// TIA Portal V18 program export: 1 tag tables, 3 data types, 7 data blocks, 7 code blocks (in call order from the OBs), 0 instance data blocks

VAR_GLOBAL   // PLC tag table "DefaultTagTable"
   convRight AT %I0.0 : Bool;
   convLeft AT %I0.1 : Bool;
   manualMode AT %Q0.2 : Bool;
   automaticMode AT %Q0.3 : Bool;
END_VAR

TYPE "typeConvCmd"
TITLE = Conveyor command
VERSION : 0.1
//input Signals to Conv
   STRUCT
      enable : Bool;
      inputLigBeam : Bool;   // light beam on input of conveyor
      editLigBeam : Bool;   // light beam on edit station of brownie
      outputLigBeam : Bool;   // light beam on output of conveyor
      startConv : Bool;   // manual start of conveyor
      reset : Bool;   // reset of conveyor belt
      workStationDone : Bool;   // working station has done process
   END_STRUCT;

END_TYPE

TYPE "typeConvSig"
TITLE = Conveyor command / status signals
VERSION : 0.1
   STRUCT
      convIn : "typeConvCmd";
      convOut : "typeConvStat";
   END_STRUCT;

END_TYPE

TYPE "typeConvStat"
TITLE = conveyor status
VERSION : 0.1
//output signal of conveyors
   STRUCT
      valid : Bool;   // as output
      isRunning : Bool;   // conveyor is running
   END_STRUCT;

END_TYPE

DATA_BLOCK "InstConveyor"
{ S7_Optimized_Access := 'TRUE' }
VERSION : 0.1
NON_RETAIN
"Conveyor"

BEGIN

END_DATA_BLOCK

DATA_BLOCK "InstRoboter"
{ S7_Optimized_Access := 'TRUE' }
VERSION : 0.1
NON_RETAIN
"Robot"

BEGIN

END_DATA_BLOCK

DATA_BLOCK "InstSequencer"
{ S7_Optimized_Access := 'TRUE' }
VERSION : 0.1
NON_RETAIN
"Sequencer"

BEGIN
   BasicPosition.T_MAX := T#0MS;
   BasicPosition.T_WARN := T#0MS;
   StartConveyor.T_MAX := T#420MS;
   StartConveyor.T_WARN := T#385MS;
   MovePart.T_MAX := T#6S_408MS;
   MovePart.T_WARN := T#5S_874MS;
   GoToStation.T_MAX := T#3S_936MS;
   GoToStation.T_WARN := T#3S_608MS;
   Fill.T_MAX := T#3S_606MS;
   Fill.T_WARN := T#3S_305MS;
   GoToMagazine.T_MAX := T#3S_966MS;
   GoToMagazine.T_WARN := T#3S_635MS;
   RemovePart.T_MAX := T#4S_56MS;
   RemovePart.T_WARN := T#3S_718MS;
   ResetPositions.T_MAX := T#0MS;
   ResetPositions.T_WARN := T#0MS;
   ResetConveyor.T_MAX := T#0MS;
   ResetConveyor.T_WARN := T#0MS;

END_DATA_BLOCK

DATA_BLOCK "InstSimulation"
{ S7_Optimized_Access := 'TRUE' }
VERSION : 0.1
NON_RETAIN
"Simulation"

BEGIN

END_DATA_BLOCK

DATA_BLOCK "SeqData"
{ S7_Optimized_Access := 'TRUE' }
VERSION : 0.1
NON_RETAIN
   VAR 
      startButton : Bool;   // Start sequence
      ackSeq : Bool;   // Acknowledge sequence errors
      switchOffSeq : Bool;   // Stop sequence
      initSeq : Bool;   // Initialise sequence
      simulateError : Bool;   // Engine has fault (simulated)
      resetCrit : Bool;   // Reset sequence errors
      seqNumber : Int;   // Active sequence number
      error : Bool;   // Sequence has an error
      automaticMode : Bool;   // Sequence mode: automatic
      manualMode : Bool;   // Sequence mode: manual
      lightBeam1 : Bool;
      lightBeam2 : Bool;
      lightBeam3 : Bool;
      partInPos1 : Bool;   // Status part is in position 1
      partInPos2 : Bool;   // Status part is in position 2
      partInPos3 : Bool;   // Status part is in position 3
      robotFill : Bool;   // Command for robot to fill part
      robotGoToStation : Bool;   // Command for robot to go to station
      robotGoToMagazine : Bool;   // Command for robot to go to magazine
      robotOnStation : Bool;   // Status robot is on station
      robotOnMagazine : Bool;   // Status robot is on magazine
      startConv : Bool;   // Command for conveyor to run
      mySupervision : Bool;   // My Supervision
      myInterlock : Bool;   // My Interlock
   END_VAR


BEGIN
   startButton := false;
   partInPos1 := false;
   myInterlock := true;

END_DATA_BLOCK

DATA_BLOCK "SimulationData"
{ S7_Optimized_Access := 'TRUE' }
VERSION : 0.1
NON_RETAIN
   VAR 
      xPos : Int;   // I
      yPos : Int;   // I
      lightBeam1 : Bool;   // I
      lightBeam2 : Bool;   // I
      lightBeam3 : Bool;   // I
      robotArmUp : Bool;   // Q
      robotArmDown : Bool;   // Q
      robotArmLeft : Bool;   // Q
      robotArmRight : Bool;   // Q
      press : Bool;   // Q
      conveyorRight : Bool;   // Q
      robotPosHMI : Int;
      robotHasChip : Bool;
   END_VAR


BEGIN

END_DATA_BLOCK

DATA_BLOCK "extension block_DB"
{ DB_Accessible_From_OPC_UA := 'FALSE' ;
 S7_Optimized_Access := 'TRUE' }
VERSION : 0.1
NON_RETAIN
"extension block"

BEGIN

END_DATA_BLOCK

ORGANIZATION_BLOCK "Main"   // OB1, LAD, ProgramCycle
TITLE = "Main Program Sweep (Cycle)"
{ S7_Optimized_Access := 'TRUE' }
VERSION : 0.1
// stored: AutoNumber true, IsIECCheckEnabled true, SetENOAutomatically false
   VAR_INPUT
      Initial_Call : Bool;   // Initial call of this OB
      Remanence : Bool;   // =True, if remanent data are available
   END_VAR
BEGIN

REGION Network 1: call conveyor
   // //=============================================================================
   // //Siemens AG // (c)Copyright (2018)
   // //-----------------------------------------------------------------------------
   // // Library: (that the source is dedicated to)
   // // Tested with: (test system with FW version)
   // // Engineering: TIA Portal V15
   // // Restrictions: (OB types, etc.)
   // // Requirements: (hardware, technological package, memory needed, etc.)
   // // Functionality: (that is implemented in the block)
   // //-----------------------------------------------------------------------------
   // // Change log table:
   // // Version Date Expert in charge Changes applied
   // // 24.08.18 dd.mm.yyyy (Name of expert) First released version
   // //=============================================================================
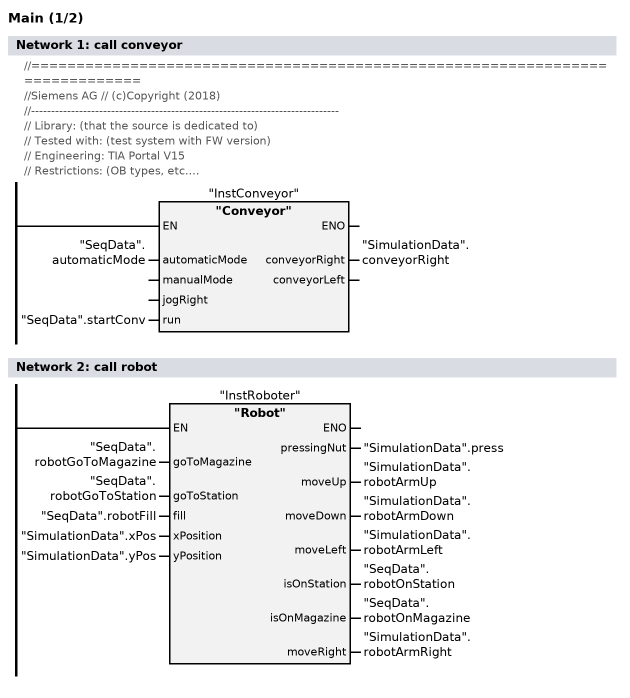
   RUNG wire#powerrail
      "InstConveyor"(automaticMode := "SeqData".automaticMode, manualMode :=, jogRight :=, run := "SeqData".startConv, conveyorRight => "SimulationData".conveyorRight, conveyorLeft =>)
   END_RUNG
   // the same network as SCL:
   "InstConveyor"(automaticMode := "SeqData".automaticMode,   // "Conveyor"
                  run := "SeqData".startConv,
                  conveyorRight => "SimulationData".conveyorRight);
END_REGION

REGION Network 2: call robot
   RUNG wire#powerrail
      "InstRoboter"(goToMagazine := "SeqData".robotGoToMagazine, goToStation := "SeqData".robotGoToStation, fill := "SeqData".robotFill, xPosition := "SimulationData".xPos, yPosition := "SimulationData".yPos, pressingNut => "SimulationData".press, moveUp => "SimulationData".robotArmUp, moveDown => "SimulationData".robotArmDown, moveLeft => "SimulationData".robotArmLeft, isOnStation => "SeqData".robotOnStation, isOnMagazine => "SeqData".robotOnMagazine, moveRight => "SimulationData".robotArmRight)
   END_RUNG
   // the same network as SCL:
   "InstRoboter"(goToMagazine := "SeqData".robotGoToMagazine,   // "Robot"
                 goToStation := "SeqData".robotGoToStation,
                 fill := "SeqData".robotFill,
                 xPosition := "SimulationData".xPos,
                 yPosition := "SimulationData".yPos,
                 pressingNut => "SimulationData".press,
                 moveUp => "SimulationData".robotArmUp,
                 moveDown => "SimulationData".robotArmDown,
                 moveLeft => "SimulationData".robotArmLeft,
                 isOnStation => "SeqData".robotOnStation,
                 isOnMagazine => "SeqData".robotOnMagazine,
                 moveRight => "SimulationData".robotArmRight);
END_REGION

REGION Network 3: call sequencer
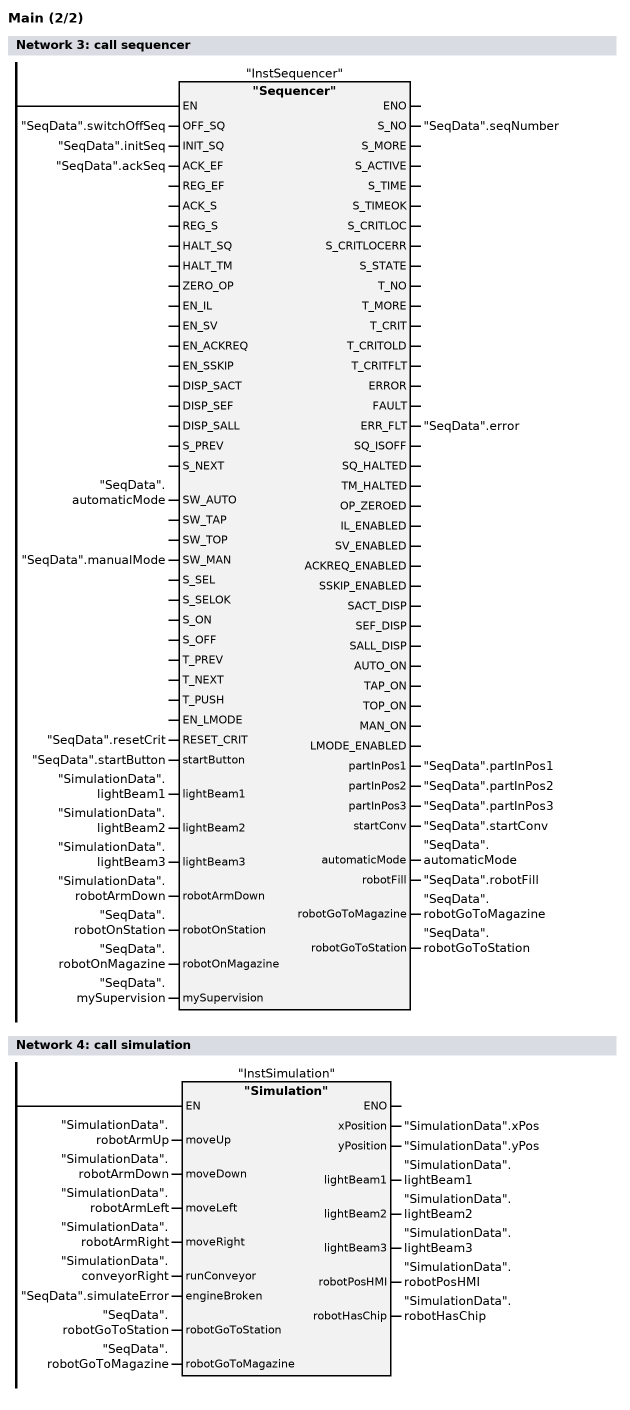
   RUNG wire#powerrail
      "InstSequencer"(OFF_SQ := "SeqData".switchOffSeq, INIT_SQ := "SeqData".initSeq, ACK_EF := "SeqData".ackSeq, REG_EF :=, ACK_S :=, REG_S :=, HALT_SQ :=, HALT_TM :=, ZERO_OP :=, EN_IL :=, EN_SV :=, EN_ACKREQ :=, EN_SSKIP :=, DISP_SACT :=, DISP_SEF :=, DISP_SALL :=, S_PREV :=, S_NEXT :=, SW_AUTO := "SeqData".automaticMode, SW_TAP :=, SW_TOP :=, SW_MAN := "SeqData".manualMode, S_SEL :=, S_SELOK :=, S_ON :=, S_OFF :=, T_PREV :=, T_NEXT :=, T_PUSH :=, EN_LMODE :=, RESET_CRIT := "SeqData".resetCrit, startButton := "SeqData".startButton, lightBeam1 := "SimulationData".lightBeam1, lightBeam2 := "SimulationData".lightBeam2, lightBeam3 := "SimulationData".lightBeam3, robotArmDown := "SimulationData".robotArmDown, robotOnStation := "SeqData".robotOnStation, robotOnMagazine := "SeqData".robotOnMagazine, mySupervision := "SeqData".mySupervision, S_NO => "SeqData".seqNumber, S_MORE =>, S_ACTIVE =>, S_TIME =>, S_TIMEOK =>, S_CRITLOC =>, S_CRITLOCERR =>, S_STATE =>, T_NO =>, T_MORE =>, T_CRIT =>, T_CRITOLD =>, T_CRITFLT =>, ERROR =>, FAULT =>, ERR_FLT => "SeqData".error, SQ_ISOFF =>, SQ_HALTED =>, TM_HALTED =>, OP_ZEROED =>, IL_ENABLED =>, SV_ENABLED =>, ACKREQ_ENABLED =>, SSKIP_ENABLED =>, SACT_DISP =>, SEF_DISP =>, SALL_DISP =>, AUTO_ON =>, TAP_ON =>, TOP_ON =>, MAN_ON =>, LMODE_ENABLED =>, partInPos1 => "SeqData".partInPos1, partInPos2 => "SeqData".partInPos2, partInPos3 => "SeqData".partInPos3, startConv => "SeqData".startConv, automaticMode => "SeqData".automaticMode, robotFill => "SeqData".robotFill, robotGoToMagazine => "SeqData".robotGoToMagazine, robotGoToStation => "SeqData".robotGoToStation)
   END_RUNG
   // the same network as SCL:
   "InstSequencer"(OFF_SQ := "SeqData".switchOffSeq,   // "Sequencer"
                   INIT_SQ := "SeqData".initSeq,
                   ACK_EF := "SeqData".ackSeq,
                   SW_AUTO := "SeqData".automaticMode,
                   SW_MAN := "SeqData".manualMode,
                   RESET_CRIT := "SeqData".resetCrit,
                   startButton := "SeqData".startButton,
                   lightBeam1 := "SimulationData".lightBeam1,
                   lightBeam2 := "SimulationData".lightBeam2,
                   lightBeam3 := "SimulationData".lightBeam3,
                   robotArmDown := "SimulationData".robotArmDown,
                   robotOnStation := "SeqData".robotOnStation,
                   robotOnMagazine := "SeqData".robotOnMagazine,
                   mySupervision := "SeqData".mySupervision,
                   S_NO => "SeqData".seqNumber,
                   ERR_FLT => "SeqData".error,
                   partInPos1 => "SeqData".partInPos1,
                   partInPos2 => "SeqData".partInPos2,
                   partInPos3 => "SeqData".partInPos3,
                   startConv => "SeqData".startConv,
                   automaticMode => "SeqData".automaticMode,
                   robotFill => "SeqData".robotFill,
                   robotGoToMagazine => "SeqData".robotGoToMagazine,
                   robotGoToStation => "SeqData".robotGoToStation);
END_REGION

REGION Network 4: call simulation
   RUNG wire#powerrail
      "InstSimulation"(moveUp := "SimulationData".robotArmUp, moveDown := "SimulationData".robotArmDown, moveLeft := "SimulationData".robotArmLeft, moveRight := "SimulationData".robotArmRight, runConveyor := "SimulationData".conveyorRight, engineBroken := "SeqData".simulateError, robotGoToStation := "SeqData".robotGoToStation, robotGoToMagazine := "SeqData".robotGoToMagazine, xPosition => "SimulationData".xPos, yPosition => "SimulationData".yPos, lightBeam1 => "SimulationData".lightBeam1, lightBeam2 => "SimulationData".lightBeam2, lightBeam3 => "SimulationData".lightBeam3, robotPosHMI => "SimulationData".robotPosHMI, robotHasChip => "SimulationData".robotHasChip)
   END_RUNG
   // the same network as SCL:
   "InstSimulation"(moveUp := "SimulationData".robotArmUp,   // "Simulation"
                    moveDown := "SimulationData".robotArmDown,
                    moveLeft := "SimulationData".robotArmLeft,
                    moveRight := "SimulationData".robotArmRight,
                    runConveyor := "SimulationData".conveyorRight,
                    engineBroken := "SeqData".simulateError,
                    robotGoToStation := "SeqData".robotGoToStation,
                    robotGoToMagazine := "SeqData".robotGoToMagazine,
                    xPosition => "SimulationData".xPos,
                    yPosition => "SimulationData".yPos,
                    lightBeam1 => "SimulationData".lightBeam1,
                    lightBeam2 => "SimulationData".lightBeam2,
                    lightBeam3 => "SimulationData".lightBeam3,
                    robotPosHMI => "SimulationData".robotPosHMI,
                    robotHasChip => "SimulationData".robotHasChip);
END_REGION
END_ORGANIZATION_BLOCK

FUNCTION_BLOCK "Conveyor"   // FB2, FBD
{ S7_Optimized_Access := 'TRUE' }
VERSION : 0.1
// stored: AutoNumber true, IsIECCheckEnabled true, IsRetainMemResEnabled false, MemoryReserve 100, SetENOAutomatically false, UDAEnableTagReadback false
   VAR_INPUT
      automaticMode : Bool;
      manualMode : Bool;
      jogRight : Bool;
      run : Bool;
   END_VAR
   VAR_OUTPUT
      conveyorRight : Bool;
      conveyorLeft : Bool;
   END_VAR
   VAR
      statRequest : Bool;
      statRelease : Bool;
   END_VAR
BEGIN

REGION Network 1 (SCL)
   //=============================================================================
   //Siemens AG // (c)Copyright (2018)
   //-----------------------------------------------------------------------------
   // Library: -
   // Tested with: CPU 1517-3 PN/DP V2.5
   // Engineering: TIA Portal V15
   // Restrictions: -
   // Requirements: PLC (S7-1500)
   // Functionality: Conveyor
   //-----------------------------------------------------------------------------
   // Change log table:
   // Version  Date      Expert in charge  Changes applied
   // 01.00.00 24.08.18  Siemens           First released version
   //=============================================================================
END_REGION

REGION Network 2
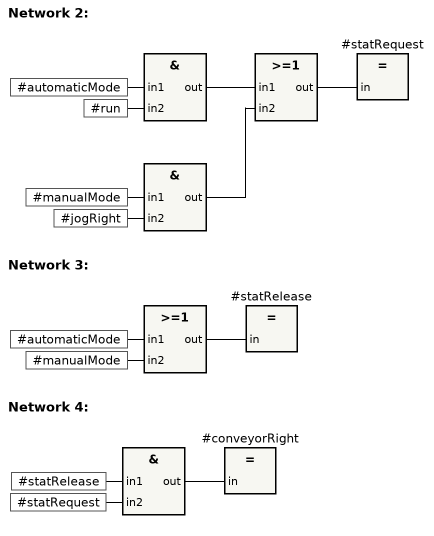
   #statRequest := (#automaticMode AND #run) OR (#manualMode AND #jogRight);
END_REGION

REGION Network 3
   #statRelease := #automaticMode OR #manualMode;
END_REGION

REGION Network 4
   #conveyorRight := #statRelease AND #statRequest;
END_REGION
END_FUNCTION_BLOCK

FUNCTION_BLOCK "Robot"
{ S7_Optimized_Access := 'TRUE' }
VERSION : 0.1
   VAR_INPUT 
      goToMagazine : Bool;
      goToStation : Bool;
      fill : Bool;
      xPosition : Int;
      yPosition : Int;
   END_VAR

   VAR_OUTPUT 
      pressingNut : Bool;
      moveUp : Bool;
      moveDown : Bool;
      moveLeft : Bool;
      isOnStation : Bool;
      isOnMagazine : Bool;
      moveRight : Bool;
   END_VAR

   VAR 
      statMoveUp : Bool;
      statMoveDown : Bool;
      statMoveLeft : Bool;
      statMoveRight : Bool;
      statIsOnMagazine : Bool;
      statPressingNut : Bool;
      statGoToStation : Bool;
      statIsOnStation : Bool;
      statRobot : Int;
   END_VAR

   VAR_TEMP 
      tempYPosition : Int;
      tempXPosition : Int;
   END_VAR

   VAR CONSTANT 
      ARM_UP : Int := 1;   // object arrived postion 1
      DIRECTION_RIGHT : Int := 6;
      OBJECT_FILL : Int := 4;   // object arrived postion 2 and not filled
      DIRECTION_LEFT : Int := 2;
      ARM_DOWN : Int := 3;   // object arrived postion 2 and filled
      ARM_UP_BACK : Int := 5;
      ARM_DOWN_BACK : Int := 7;
      IDLE : Int;
   END_VAR


BEGIN
	//=============================================================================
	//Siemens AG // (c)Copyright (2018)
	//-----------------------------------------------------------------------------
	// Library: -
	// Tested with: CPU 1517-3 PN/DP V2.5
	// Engineering: TIA Portal V15
	// Restrictions: -
	// Requirements: PLC (S7-1500)
	// Functionality: Robot
	//-----------------------------------------------------------------------------
	// Change log table:
	// Version  Date      Expert in charge  Changes applied
	// 01.00.00 24.08.18  Siemens           First released version
	//=============================================================================
	
	// read inputs
	#tempYPosition := #yPosition;
	#tempXPosition := #xPosition;
	
	CASE #statRobot OF
	    //robot on magazine   
	  #IDLE:
	    #statMoveDown := FALSE;
	    #statIsOnMagazine := FALSE;
	    IF (#goToStation = TRUE)
	    THEN
	      #statRobot := #ARM_UP;
	    END_IF;
	    
	    //robot moves up 
	  #ARM_UP:
	    #statMoveDown := FALSE;
	    #statMoveUp := TRUE;
	    IF (#tempYPosition = 100)
	    THEN
	      #statRobot := #DIRECTION_LEFT;
	    END_IF;
	    
	    //robot moves to the left direction     
	  #DIRECTION_LEFT:
	    #statMoveUp := FALSE;
	    #statMoveLeft := TRUE;
	    IF (#tempXPosition = 100)
	    THEN
	      #statRobot := #ARM_DOWN
	      ;
	    END_IF;
	    
	    //robot moves down    
	  #ARM_DOWN:
	    #statMoveLeft := FALSE;
	    #statMoveDown := TRUE;
	    IF (#tempYPosition = 0)
	    THEN
	      #statIsOnStation := TRUE;
	      #statRobot := #OBJECT_FILL;
	    END_IF;
	    
	    //fill  
	  #OBJECT_FILL:
	    #statMoveDown := FALSE;
	    #statIsOnStation := FALSE;
	    #statPressingNut := #fill;
	    IF (#goToMagazine = TRUE)
	    THEN
	      #statRobot := #ARM_UP_BACK;
	    END_IF;
	    
	    //robot moves up 
	  #ARM_UP_BACK:
	    #statMoveUp := TRUE;
	    #statPressingNut := FALSE;
	    IF (#tempYPosition = 100)
	    THEN
	      #statRobot := #DIRECTION_RIGHT;
	    END_IF;
	    
	    //robot moves to the right direction     
	  #DIRECTION_RIGHT:
	    #statMoveUp := FALSE;
	    #statMoveRight := TRUE;
	    IF (#tempXPosition = 0)
	    THEN
	      #statRobot := #ARM_DOWN_BACK;
	    END_IF;
	    
	    //robot moves down back to magazine    
	  #ARM_DOWN_BACK:
	    #statMoveRight := FALSE;
	    #statMoveDown := TRUE;
	    IF (#tempYPosition = 0)
	    THEN
	      #statIsOnMagazine := TRUE;
	      #statRobot := #IDLE;
	    END_IF;
	    
	  ELSE  // Statement section ELSE
	    ;
	END_CASE;
	
	//write outputs
	#moveUp := #statMoveUp;
	#moveDown := #statMoveDown;
	#moveLeft := #statMoveLeft;
	#moveRight := #statMoveRight;
	#isOnMagazine := #statIsOnMagazine;
	#isOnStation := #statIsOnStation;
	#pressingNut := #statPressingNut;
	
END_FUNCTION_BLOCK

FUNCTION_BLOCK "Sequencer"   // FB4, GRAPH
VERSION : 0.1
// stored: AcknowledgeErrorsRequired true, AutoNumber true, ExtensionBlockName "ExtensionToGRAPH", GraphVersion 5.0, InitialValuesAcquisition true, IsIECCheckEnabled true, LanguageInNetworks FBD, LockOperatingMode false, PermanentILProcessingInMANMode false, SetENOAutomatically false, SkipSteps false, UDAEnableTagReadback false, WithAlarmHandling true
   // inherited from GRAPH_BASE
   VAR
      OFF_SQ_BASE : Bool;
   END_VAR
   VAR_INPUT
      OFF_SQ { ExternalWritable := 'False'} : Bool := false;   // Kette ausschalten / Turn sequence off / Désactiver le graphe
      INIT_SQ { ExternalWritable := 'False'} : Bool := false;   // Kette in Initialzustand versetzen
      ACK_EF { ExternalWritable := 'False'} : Bool := false;   // Alle Fehler und Störungen quittieren / Acknowledge all errors and faults / Acquitter toutes les erreurs et perturbations
      REG_EF { ExternalWritable := 'False'} : Bool := false;   // Alle Fehler und Störungen registrieren / Register all errors and faults / Enregistrer toutes les erreurs et perturbations
      ACK_S { ExternalWritable := 'False'} : Bool := false;   // Schritt quittieren, der an Parameter S_NO anliegt / Acknowledge step indicated in S_NO / Acquitter l'étape figurant dans le paramètre S_NO
      REG_S { ExternalWritable := 'False'} : Bool := false;   // Schritt registrieren, der an Parameter S_NO anliegt / Register the step indicated in S_NO / Enregistrer l'étape figurant dans le paramètre S_NO
      HALT_SQ { ExternalWritable := 'False'} : Bool := false;   // Kette sofort anhalten / Halt sequence immediately / Arrêter le graphe immédiatement
      HALT_TM { ExternalWritable := 'False'} : Bool := false;   // Zeiten sofort anhalten / Halt timers immediately / Arrêter les temporisations immédiatement
      ZERO_OP { ExternalWritable := 'False'} : Bool := false;   // Alle mit N, L, D zugewiesenen Operanden auf 0 setzen / Set all operands assigned with N, L, D to 0 / Mettre à 0 tous les opérandes affectés avec N, L, D
      EN_IL { ExternalWritable := 'False'} : Bool := false;   // Interlockbearbeitung aktivieren / Activate interlocks / Activer le traitement des Interlocks
      EN_SV { ExternalWritable := 'False'} : Bool := false;   // Supervisionsbearbeitung aktivieren / Activate supervision processing / Activer le traitement de Supervision
      EN_ACKREQ { ExternalWritable := 'False'} : Bool := false;   // Quittierpflicht aktivieren / Activate mandatory acknowledgment / Activer l'obligation d'acquittement
      EN_SSKIP { ExternalWritable := 'False'} : Bool := false;   // "Schritte überspringen" aktivieren / Enable "Skip step" / Activer "Ignorer l'étape"
      DISP_SACT { ExternalWritable := 'False'} : Bool := false;   // Nur aktive Schritte anzeigen / Display active steps only / Afficher uniquement les étapes activées
      DISP_SEF { ExternalWritable := 'False'} : Bool := false;   // Nur fehlerhafte und gestörte Schritte anzeigen / Display only steps with errors and disrupted steps / Afficher uniquement les étapes avec erreurs et perturbations
      DISP_SALL { ExternalWritable := 'False'} : Bool := false;   // Alle Schritte anzeigen / Display all steps / Afficher toutes les étapes
      S_PREV { ExternalWritable := 'False'} : Bool := false;   // Vorherigen Schritt am Parameter S_NO ausgeben / Output previous step in parameter S_NO / Afficher l'étape précédente dans le paramètre S_NO
      S_NEXT { ExternalWritable := 'False'} : Bool := false;   // Nächsten Schritt am Parameter S_NO anzeigen / Indicate next step in parameter S_NO / Afficher l'étape suivante dans le paramètre S_NO
      SW_AUTO { ExternalWritable := 'False'} : Bool := false;   // Automatischer Betrieb / Automatic mode / Mode automatique
      SW_TAP { ExternalWritable := 'False'} : Bool := false;   // Halbautomatisch/Weiterschalten mit Transition / Semiautomatic/switch with transition / Mode semi-automatique/Activation de l'étape suivante avec transition
      SW_TOP { ExternalWritable := 'False'} : Bool := false;   // Halbautomatisch/Ignoriere Transition / Semiautomatic/ignore transition / Mode semi-automatique/Ignorer la transition
      SW_MAN { ExternalWritable := 'False'} : Bool := false;   // Handbetrieb / Manual mode / Mode manuel
      S_SEL { ExternalWritable := 'False'} : Int := 0;   // Schritt auswählen, der an S_NO ausgegeben werden soll / Select step to be output to S_NO / Sélectionner l'étape à afficher dans S_NO
      S_SELOK { ExternalWritable := 'False'} : Bool := false;   // Wert aus S_SEL nach S_NO übernehmen / Enter value from S_SEL in S_NO / Appliquer la valeur de S_SEL à S_NO
      S_ON { ExternalWritable := 'False'} : Bool := false;   // Schritt aktivieren, der an Parameter S_NO anliegt / Activate step indicated in S_NO / Activer l'étape figurant dans le paramètre S_NO
      S_OFF { ExternalWritable := 'False'} : Bool := false;   // Schritt deaktivieren, der an Parameter S_NO anliegt / Deactivate step indicated S_NO / Désactiver l'étape figurant dans le paramètre S_NO
      T_PREV { ExternalWritable := 'False'} : Bool := false;   // Vorherige Transition an Parameter T_NO anzeigen / Display previous transition in T_NO / Afficher la transition précédente dans le paramètre T_NO
      T_NEXT { ExternalWritable := 'False'} : Bool := false;   // Nächste Transition an Parameter T_NO anzeigen / Display next transition at parameter T_NO / Afficher la transition suivante dans le paramètre T_NO
      T_PUSH { ExternalWritable := 'False'} : Bool := false;   // Schaltfreigabe für Transition im halbautomatischen Betrieb / Enable transition to switch in semi automatic mode / Validation de commutation pour transition en mode semi-automatique
      EN_LMODE { ExternalWritable := 'False'} : Bool := false;   // Lernmodus aktivieren / Activate learning mode / Activer le mode apprentissage
      RESET_CRIT { ExternalWritable := 'False'} : Bool := false;   // Alle Erstwerte, die für Interlocks und Transitionen aufgezeichnet wurden, zurücksetzen / Reset all initial values recorded for interlocks and transitions / Réinitialiser toutes les premières valeurs enregistrées pour les Interlocks et les transitions
      startButton : Bool;
      lightBeam1 : Bool;
      lightBeam2 : Bool;
      lightBeam3 : Bool;
      robotArmDown : Bool;
      robotOnStation : Bool;
      robotOnMagazine : Bool;
      mySupervision : Bool;
   END_VAR
   VAR_OUTPUT
      S_NO { ExternalWritable := 'False'} : Int := 0;   // Schrittnummer / Step number / Numéro d'étape
      S_MORE { ExternalWritable := 'False'} : Bool := false;   // Weitere Schritte sind vorhanden und können in S_NO angezeigt werden. / More steps are available and can be shown in S_NO / Il existe d'autres étapes qui peuvent être affichées dans S_NO.
      S_ACTIVE { ExternalWritable := 'False'} : Bool := false;   // Schritt, der an Parameter S_NO angezeigt wird, ist aktiv / Step indicated in S_NO is active / L'étape affichée dans le paramètre S_NO est activée
      S_TIME { ExternalWritable := 'False'} : Time := T#0ms;   // Schrittaktivierungszeit / Step activation time / Temps d'activation d'étape
      S_TIMEOK { ExternalWritable := 'False'} : Time := T#0ms;   // Schrittaktivierungszeit fehlerfrei / No error in step activation time / Temps d'activation d'étape sans erreur
      S_CRITLOC { ExternalWritable := 'False'} : DWord := 16#0;   // Interlock-Kriterienbits / Interlock criteria bits / Bits de critère Interlock
      S_CRITLOCERR { ExternalWritable := 'False'} : DWord := 16#0;   // Interlock-Kriterienbits bei Ereignis L1 / Interlock criteria bits for event L1 / Bits de critère Interlock pour l'événement L1
      S_STATE { ExternalWritable := 'False'} : Word := 16#0;   // Schrittzustandsbits / Step state bits / Bits d'état d'étape
      T_NO { ExternalWritable := 'False'} : Int := 0;   // Transitionsnummer / Transition number / Numéro de transition
      T_MORE { ExternalWritable := 'False'} : Bool := false;   // Weitere gültige Transitionen zur Anzeige verfügbar / More valid transitions available for display / D'autres transitions valides sont disponibles pour affichage
      T_CRIT { ExternalWritable := 'False'} : DWord := 16#0;   // Transitions-Kriterienbits / Transition criteria bits / Bits de critère de transition
      T_CRITOLD { ExternalWritable := 'False'} : DWord := 16#0;   // Transitions-Kriterienbits des letzten Zyklus / Transition criteria bits from last cycle / Bits de critère de transition du dernier cycle
      T_CRITFLT { ExternalWritable := 'False'} : DWord := 16#0;   // Transitions-Kriterienbits bei Ereignis V1 / Transition criteria bits for event V1 / Bits de critère de transition pour l'événement V1
      ERROR { ExternalWritable := 'False'} : Bool := false;   // Sammelfehler Interlock / Interlock group error / Erreur groupée Interlock
      FAULT { ExternalWritable := 'False'} : Bool := false;   // Sammelfehler Supervision / Supervision group error / Erreur groupée Supervision
      ERR_FLT { ExternalWritable := 'False'} : Bool := false;   // Sammelfehler Interlock oder Supervision / Interlock or supervision group error / Erreur groupée Interlock or Supervision
      SQ_ISOFF { ExternalWritable := 'False'} : Bool := false;   // Kette ausgeschaltet (kein Schritt aktiv) / Sequence is off (no step active) / Graphe désactivé (aucune étape n'est activée)
      SQ_HALTED { ExternalWritable := 'False'} : Bool := false;   // Kette angehalten / Sequence halted / Graphe arrêté
      TM_HALTED { ExternalWritable := 'False'} : Bool := false;   // Zeiten angehalten / Timers halted / Les temporisations sont arrêtées
      OP_ZEROED { ExternalWritable := 'False'} : Bool := false;   // Alle mit N, L oder D zugewiesenen Operanden auf 0 gesetzt / All the operands assigned with N, L, D are set to 0 / Tous les opérandes affectés avec N, L ou D sont mis à 0
      IL_ENABLED { ExternalWritable := 'False'} : Bool := false;   // Interlockbearbeitung aktiv / Interlocks are active / Traitement des Interlocks activé
      SV_ENABLED { ExternalWritable := 'False'} : Bool := false;   // Supervisionsbearbeitung aktiviert / Supervision processing activated / Traitement de Supervision activé
      ACKREQ_ENABLED { ExternalWritable := 'False'} : Bool := false;   // Quittierpflicht aktiviert / Mandatory acknowledgment activated / Obligation d'acquittement activée
      SSKIP_ENABLED { ExternalWritable := 'False'} : Bool := false;   // Schritte überspringen aktiviert / Skip steps activated / Ignorer les étapes activé
      SACT_DISP { ExternalWritable := 'False'} : Bool := false;   // Nur aktive Schritte anzeigen / Display active steps only / Afficher uniquement les étapes activées
      SEF_DISP { ExternalWritable := 'False'} : Bool := false;   // Nur fehlerhafte oder gestörte Schritte anzeigen / Display only steps with errors or disrupted steps / Afficher uniquement les étapes avec erreurs ou perturbations
      SALL_DISP { ExternalWritable := 'False'} : Bool := false;   // Alle Schritte anzeigen / Display all steps / Afficher toutes les étapes
      AUTO_ON { ExternalWritable := 'False'} : Bool := false;   // Automatischer Betrieb eingeschaltet / Automatic mode is active / Mode automatique activé
      TAP_ON { ExternalWritable := 'False'} : Bool := false;   // Halbautomatischer Betrieb/Schritt mit Transition eingeschaltet / Semiautomatic mode/step with transition enabled / Mode semi-automatique/Etape avec transition activé
      TOP_ON { ExternalWritable := 'False'} : Bool := false;   // Halbautomatischer Betrieb/Ignoriere Transition eingeschaltet / Semiautomatic mode/ignore transition enabled / Mode semi-automatique/Ignorer la transition activé
      MAN_ON { ExternalWritable := 'False'} : Bool := false;   // Handbetrieb eingeschaltet / Manual mode is active / Mode manuel activé
      LMODE_ENABLED { ExternalWritable := 'False'} : Bool := false;   // Lernmodus aktiv / Learning mode is active / Mode apprentissage actif
      partInPos1 : Bool;
      partInPos2 : Bool;
      partInPos3 : Bool;
      startConv : Bool;
      automaticMode : Bool;
      robotFill : Bool;
      robotGoToMagazine : Bool;
      robotGoToStation : Bool;
   END_VAR
   VAR
      statLightbeam3Fal : Bool;
      statMemoryTag : Bool;
      instExtensionToGRAPH { S7_SetPoint := 'True'} : "ExtensionToGRAPH";
      memTag { ExternalAccessible := 'False'; ExternalVisible := 'False'; ExternalWritable := 'False'} : Bool;
      lightBeam3Fall { ExternalAccessible := 'False'; ExternalVisible := 'False'; ExternalWritable := 'False'} : Bool;
      out1 { ExternalAccessible := 'False'; ExternalVisible := 'False'; ExternalWritable := 'False'} : Bool;
      safetyOK { ExternalAccessible := 'False'; ExternalVisible := 'False'; ExternalWritable := 'False'} : Bool;
   END_VAR
   VAR_TEMP
      tagError : Int;
      dateTime : Date_And_Time;
      retval : Time;
      timeTick : Time;
      minLimit : Real;
      inReal : Real;
      maxLimit : Real;
      outReal : Real;
      in1 : Bool;
      in2 : Bool;
   END_VAR
   VAR_TEMP   // added for the SCL form of the ladder/FBD networks
      _w1 : Bool;
   END_VAR
BEGIN
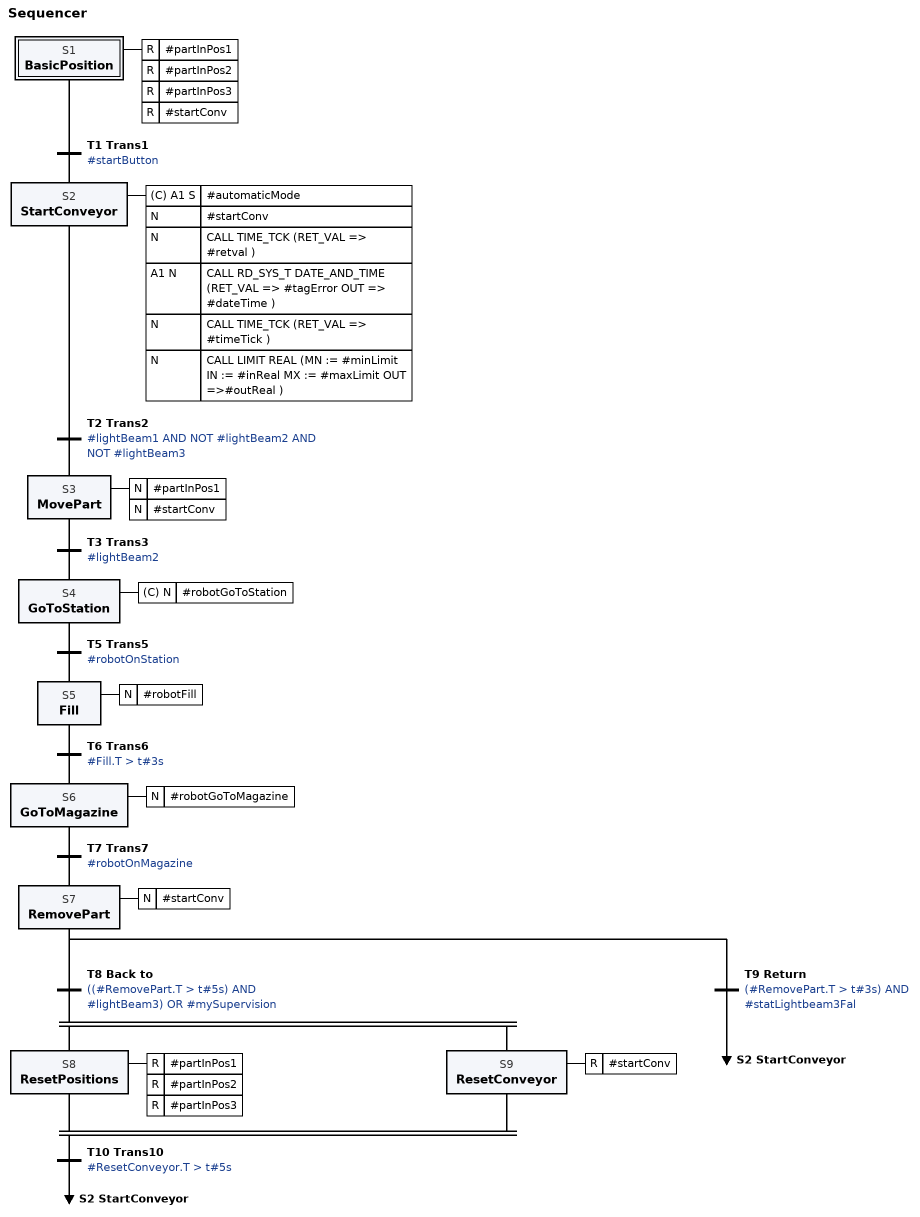
   // permanent pre-instructions
   NETWORK 1
   TITLE = comment 1
      #_w1 := NOT "SimulationData".lightBeam3 AND #memTag;   // falling edge of "SimulationData".lightBeam3
      #memTag := "SimulationData".lightBeam3;
      #lightBeam3Fall := #_w1;
   NETWORK 2
   TITLE = comment 2
      #out1 := NOT (#in1 AND #in2);
   NETWORK 3
   TITLE = comment 2
      #out1 := NOT (#in1 XOR #in2);

   // sequencer 1
   // //=============================================================================
   // //Siemens AG // (c)Copyright (2018)
   // //-----------------------------------------------------------------------------
   // // Library: -
   // // Tested with: CPU 1517-3 PN/DP V2.5
   // // Engineering: TIA Portal V15
   // // Restrictions: -
   // // Requirements: PLC (S7-1500)
   // // Functionality: Sequencer
   // //-----------------------------------------------------------------------------
   // // Change log table:
   // // Version    Date         Expert in charge  Changes applied
   // // 01.00.00 24.08.18  Siemens                First released version
   // //=============================================================================
   INITIAL_STEP BasicPosition:   // S1, max time T#10S, warning time T#7S
      interlock C := (none);   // safety not OK
              R    #partInPos1
              R    #partInPos2
              R    #partInPos3
              R    #startConv
   END_STEP
   TRANSITION Trans1 FROM BasicPosition TO StartConveyor   // T1
      := #startButton;
   END_TRANSITION
   STEP StartConveyor:   // S2, max time T#10S, warning time T#7S
      (C) A1  S    #automaticMode
              N    #startConv
              N    CALL TIME_TCK
                   (RET_VAL => #retval
                   )
          A1  N    CALL RD_SYS_T DATE_AND_TIME
                   (RET_VAL => #tagError
                   OUT => #dateTime
                   )
              N    CALL TIME_TCK
                   (RET_VAL => #timeTick
                   )
              N    CALL LIMIT REAL
                   (MN := #minLimit
                   IN := #inReal
                   MX := #maxLimit
                   OUT =>#outReal
                   )
   END_STEP
   TRANSITION Trans2 FROM StartConveyor TO MovePart   // T2
      := #lightBeam1 AND NOT #lightBeam2 AND NOT #lightBeam3;
   END_TRANSITION
   STEP MovePart:   // S3, max time T#10S, warning time T#7S
      supervision V := (none);   // Schrittaktivierungszeit überschritten / Step activation time is exceeded
              N    #partInPos1
              N    #startConv
   END_STEP
   TRANSITION Trans3 FROM MovePart TO GoToStation   // T3
      := #lightBeam2;
   END_TRANSITION
   STEP GoToStation:   // S4, max time T#10S, warning time T#7S
      interlock C := NOT #robotArmDown;   // Robot is up
      (C)     N    #robotGoToStation
   END_STEP
   TRANSITION Trans5 FROM GoToStation TO Fill   // T5
      := #robotOnStation;
   END_TRANSITION
   STEP Fill:   // S5, max time T#10S, warning time T#7S
              N    #robotFill
   END_STEP
   TRANSITION Trans6 FROM Fill TO GoToMagazine   // T6
      := #Fill.T > t#3s;
   END_TRANSITION
   STEP GoToMagazine:   // S6, max time T#10S, warning time T#7S
              N    #robotGoToMagazine
   END_STEP
   TRANSITION Trans7 FROM GoToMagazine TO RemovePart   // T7
      := #robotOnMagazine;
   END_TRANSITION
   STEP RemovePart:   // S7, max time T#10S, warning time T#7S
      supervision V := (#RemovePart.T < #RemovePart.T_MAX) AND (#RemovePart.T > #RemovePart.T_WARN);   // Schrittaktivierungszeit überschritten / Step activation time is exceeded
              N    #startConv
   END_STEP
   TRANSITION "Back to" FROM RemovePart TO (ResetPositions, ResetConveyor)   // T8
      := ((#RemovePart.T > t#5s) AND #lightBeam3) OR #mySupervision;
   END_TRANSITION
   TRANSITION "Return" FROM RemovePart TO StartConveyor   // T9, jump
      := (#RemovePart.T > t#3s) AND #statLightbeam3Fal;
   END_TRANSITION
   STEP ResetPositions:   // S8, max time T#10S, warning time T#7S
      interlock C := #ResetPositions.T > #ResetPositions.T_MAX;   // Interlocks deaktivieren / Deactivate interlocks
      supervision V := (none);   // Supervision is TRUE, please set it to FALSE
              R    #partInPos1
              R    #partInPos2
              R    #partInPos3
   END_STEP
   TRANSITION Trans10 FROM (ResetConveyor, ResetPositions) TO StartConveyor   // T10, jump
      := #ResetConveyor.T > t#5s;
   END_TRANSITION
   STEP ResetConveyor:   // S9, max time T#10S, warning time T#7S
              R    #startConv
   END_STEP

   // permanent post-instructions
   NETWORK 1
      #_w1 := NOT #lightBeam3 AND #statMemoryTag;   // falling edge of #lightBeam3
      #statMemoryTag := #lightBeam3;
      #statLightbeam3Fal := #_w1;
END_FUNCTION_BLOCK

FUNCTION_BLOCK "ExtensionToGRAPH"
{ S7_Optimized_Access := 'TRUE' }
VERSION : 0.1
   VAR_IN_OUT 
      extRTData {InstructionName := 'G7_RTDataPlus_V5'; LibVersion := '1.0'} : G7_RTDataPlus_V5;   // xyz
      extG7T {InstructionName := 'G7_TransitionPlus_V5'; LibVersion := '1.0'} : Array[*] of G7_TransitionPlus_V5;
      extG7S {InstructionName := 'G7_StepPlus_V5'; LibVersion := '1.0'} : Array[*] of G7_StepPlus_V5;
      extG7Arrays : Array[*] of USInt;
   END_VAR

   VAR 
      statLowerG7T { ExternalAccessible := 'False'; ExternalVisible := 'False'; ExternalWritable := 'False'} : DInt;
      statUpperG7T { ExternalAccessible := 'False'; ExternalVisible := 'False'; ExternalWritable := 'False'} : DInt;
      statLowerG7S { ExternalAccessible := 'False'; ExternalVisible := 'False'; ExternalWritable := 'False'} : DInt;
      statUpperG7S { ExternalAccessible := 'False'; ExternalVisible := 'False'; ExternalWritable := 'False'} : DInt;
      statUserTransitionNumber : Int;
      statUserStepNumber : Int;
      statUserActiveSteps : USInt;
      statUserSatisfiedTrans : USInt;
   END_VAR

   VAR_TEMP 
      tempG7TIndex : DInt;
      tempG7SIndex : DInt;
   END_VAR


BEGIN
	//=============================================================================
	//Siemens AG // (c)Copyright (2018)
	//-----------------------------------------------------------------------------
	// Library: -
	// Tested with: CPU 1517-3 PN/DP V2.5
	// Engineering: TIA Portal V15
	// Restrictions: -
	// Requirements: PLC (S7-1500)
	// Functionality: Extension functionality for iterative access to Graph
	//                variables and invisible GraphStatusVariables.
	//-----------------------------------------------------------------------------
	// Change log table:
	// Version  Date      Expert in charge  Changes applied
	// 01.00.00 24.08.18  Siemens           First released version
	//=============================================================================
	
	REGION ReadArrayBounderies
	  
	  // Read ArrayBounderies of predefined Graph-Array's
	  #statLowerG7T := LOWER_BOUND(ARR := #extG7T, DIM := 1);
	  #statUpperG7T := UPPER_BOUND(ARR := #extG7T, DIM := 1);
	  
	  #statLowerG7S := LOWER_BOUND(ARR := #extG7S, DIM := 1);
	  #statUpperG7S := UPPER_BOUND(ARR := #extG7S, DIM := 1);
	  
	END_REGION
	
	
	REGION IterativeTransitionAccess
	  //Example: As a programmer I want to check whether a specific transition
	  //number (e.g. asked via HMI-Panel) is available in the Graph block.
	  
	  FOR #tempG7TIndex := #statLowerG7T TO #statUpperG7T BY 1 DO
	    ;
	    IF (#extG7T[#tempG7TIndex].TNO = #statUserTransitionNumber)
	    THEN
	      ;
	      // Do any action
	      // Do any action            
	    END_IF;
	  END_FOR;
	  
	END_REGION
	
	
	REGION IterativeStepAccess
	  //Example: As a programmer I want to check whether a specific step number
	  //(e.g. asked via HMI-Panel) is available in the Graph block.
	  
	  FOR #tempG7SIndex := #statLowerG7S TO #statUpperG7S BY 1 DO
	    ;
	    IF (#extG7S[#tempG7SIndex].SNO = #statUserStepNumber)
	    THEN
	      ;
	      // Do any action
	      // Do any action            
	    END_IF;
	  END_FOR;
	  
	END_REGION
	
	
	REGION ReadGraphStatusVariables
	  //*******************************************************************************************************************************************
	  //GraphStatusVariables are stored within #io_G7Array and normally invisible within the Graph block.
	  //For specific usecases the GraphStatusVariables can be used via this extension block from Graph Version V4.0 (V14 SP1).
	  //
	  //All available GraphStatusVariables are described in the online help within Chapter:
	  //"Basic information on extending the standard behavior of GRAPH"
	  //*******************************************************************************************************************************************
	  //
	  //Example 1: As a user I want to know the number of active steps "SAX" (for example: two steps are active in one cycle)
	  //
	  //         a.) Use the accumulative Array named #io_G7Array with index #io_RT_Data.OFFSETS.SAX_OFFSET
	  //         b.) #io_G7Arrays[#io_RT_Data.OFFSETS.SAX_OFFSET] give the number of the valid members within the SAX_field --> length of field
	  //             (in this example the value is 3)
	  //             #io_G7Arrays[#io_RT_Data.OFFSETS.SAX_OFFSET + 1] give the first valid index FOR active step numbers in this cycle.
	  //             #io_G7Arrays[#io_RT_Data.OFFSETS.SAX_OFFSET+2] give the second valid index for active step numbers in this cycle.
	  //             #io_G7Arrays[#io_RT_Data.OFFSETS.SAX_OFFSET+3] can be a reserve/unvalid index or already a member of the next offset.
	  //             #io_G7S[#io_G7Arrays[#io_RT_Data.OFFSETS.SAX_OFFSET + 1]].SNO give the first valid step number in this cycle.
	  //             #io_G7S[#io_G7Arrays[#io_RT_Data.OFFSETS.SAX_OFFSET + 2]].SNO give the second valid step number in this cycle.
	  //         
	  //         --> Number of active steps is "Number of valid members within SAX_field" - 1
	  
	  #statUserActiveSteps := #extG7Arrays[#extRTData.OFFSETS.SAX_OFFSET] - 1;
	  
	  
	  //Example 2: As a user I want to know the number of satisfied Transitions "TTX" (for example: one transition is satisfied within one cycle)
	  //
	  //         a.) Use the accumulative Array named #io_G7Array with index #io_RT_Data.OFFSETS.TTX_OFFSET
	  //         b.) #io_G7Arrays[#io_RT_Data.OFFSETS.TTX_OFFSET] give the number of the valid members within the TTX_field --> length of field
	  //             (in this example the value is 2)
	  //         c.) #io_G7Arrays[#io_RT_Data.OFFSETS.TTX_OFFSET+1] give the first valid index for satisfied transition numbers in this cycle.
	  //             #io_G7Arrays[#io_RT_Data.OFFSETS.TTX_OFFSET+2] can be a reserve/unvalid index or already a member of the next offset.
	  //         d.) #io_G7T[#io_G7Arrays[#io_RT_Data.OFFSETS.TTX_OFFSET + 1]].TNO give the valid transition number in this cycle.
	  //         --> Number of satisfied transitions is "Number of valid members within TTX_field" - 1
	  
	  #statUserSatisfiedTrans := #extG7Arrays[#extRTData.OFFSETS.TTX_OFFSET] - 1;
	  
	END_REGION
	
	
	
	
END_FUNCTION_BLOCK

FUNCTION_BLOCK "Simulation"   // FB6, FBD
TITLE = Simulation
{ S7_Optimized_Access := 'TRUE' }
VERSION : 0.1
// Simulates machine behavior
// stored: AutoNumber true, IsIECCheckEnabled true, IsRetainMemResEnabled false, MemoryReserve 100, SetENOAutomatically false, UDAEnableTagReadback false
   VAR_INPUT
      moveUp : Bool;
      moveDown : Bool;
      moveLeft : Bool;
      moveRight : Bool;
      runConveyor : Bool;
      engineBroken : Bool;
      robotGoToStation : Bool;
      robotGoToMagazine : Bool;
   END_VAR
   VAR_OUTPUT
      xPosition : Int;
      yPosition : Int;
      lightBeam1 : Bool;
      lightBeam2 : Bool;
      lightBeam3 : Bool;
      robotPosHMI : Int;
      robotHasChip : Bool;
   END_VAR
   VAR
      instTimerSimulate { S7_SetPoint := 'True'} : TON_TIME;
      statSimulate : Bool;
      statPositionConveyor : Int;
      statRobotHasChip : Bool;
      statRobotPosHMI : Int;
   END_VAR
   VAR_TEMP
      tempLB1 : Bool;
      tempLB2 : Bool;
      tempLB3 : Bool;
   END_VAR
   VAR CONSTANT
      SIMULATION_TIME : Time := T#10ms;
   END_VAR
BEGIN

REGION Network 1 (SCL)
   //=============================================================================
   //Siemens AG // (c)Copyright (2018)
   //-----------------------------------------------------------------------------
   // Library: -
   // Tested with: CPU 1517-3 PN/DP V2.5
   // Engineering: TIA Portal V15
   // Restrictions: -
   // Requirements: PLC (S7-1500)
   // Functionality: Simulation
   //-----------------------------------------------------------------------------
   // Change log table:
   // Version  Date      Expert in charge  Changes applied
   // 01.00.00 24.08.18  Siemens           First released version
   //=============================================================================
END_REGION

REGION Network 2: trigger simulation step
   // set bit for one cycle every 10ms
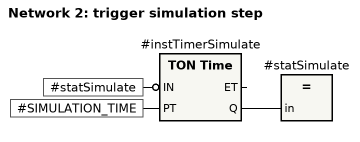
   #instTimerSimulate(IN := NOT #statSimulate, PT := #SIMULATION_TIME);   // TON
   #statSimulate := #instTimerSimulate.Q;
END_REGION

REGION Network 3 (SCL): simulation step
   //=============================================================================
   //Siemens AG // (c)Copyright (2018)
   //-----------------------------------------------------------------------------
   // Library: (that the source is dedicated to)
   // Tested with: (test system with FW version)
   // Engineering: TIA Portal V15
   // Restrictions: (OB types, etc.)
   // Requirements: (hardware, technological package, memory needed, etc.)
   // Functionality: (that is implemented in the block)
   //-----------------------------------------------------------------------------
   // Change log table:
   // Version Date Expert in charge Changes applied
   // 24.08.18 dd.mm.yyyy (Name of expert) First released version
   //=============================================================================


   IF (#statSimulate = TRUE)
     AND (NOT #engineBroken)
   THEN
     //move robot
     IF (#moveUp = TRUE)
     THEN
       #yPosition += 1;
     END_IF;
     IF (#moveDown = TRUE)
     THEN
       #yPosition -= 1;
     END_IF;
     IF (#moveLeft = TRUE)
     THEN
       #xPosition += 1;
     END_IF;
     IF (#moveRight = TRUE)
     THEN
       #xPosition -= 1;
     END_IF;
     //move conveyor
     IF (#statPositionConveyor > 800)
     THEN
       #statPositionConveyor := 0;
     ELSIF (#runConveyor = TRUE)
     THEN
       #statPositionConveyor += 1;
     END_IF;
   END_IF;

   //for S7-300 / S7-400
   #tempLB1 := FALSE;
   #tempLB2 := FALSE;
   #tempLB3 := FALSE;

   //assign lightbeams
   CASE #statPositionConveyor OF
     30..60:
       #tempLB1 := TRUE;
     500..530:
       #tempLB2 := TRUE;
     780..800:
       #tempLB3 := TRUE;

     ELSE  // Statement section ELSE
       ;
   END_CASE;

   #lightBeam1 := #tempLB1;
   #lightBeam2 := #tempLB2;
   #lightBeam3 := #tempLB3;

   //Calculate data for display of robot in HMI
   IF (#xPosition = 100)
   THEN
     #statRobotPosHMI := #yPosition;
   ELSE
       #statRobotPosHMI :=100;
   END_IF;

   IF (#robotGoToStation)
   THEN
       #statRobotHasChip := TRUE;
   END_IF;
   IF (#robotGoToMagazine = TRUE)
     OR (#statRobotPosHMI = 0)
   THEN
     #statRobotHasChip := FALSE;
   END_IF;

   // wirte outputs
   #robotHasChip:= #statRobotHasChip;
   #robotPosHMI := #statRobotPosHMI;
END_REGION
END_FUNCTION_BLOCK

FUNCTION_BLOCK "extension block"
{ S7_Optimized_Access := 'TRUE' }
VERSION : 0.1
   VAR_IN_OUT 
      InOutRTData {InstructionName := 'G7_RTDataPlus_V5'; LibVersion := '1.0'} : G7_RTDataPlus_V5;
      InOutG7T {InstructionName := 'G7_TransitionPlus_V5'; LibVersion := '1.0'} : Array[*] of G7_TransitionPlus_V5;
      InOutG7S {InstructionName := 'G7_StepPlus_V5'; LibVersion := '1.0'} : Array[*] of G7_StepPlus_V5;
      InOutG7Arrays : Array[*] of USInt;
   END_VAR

   VAR_TEMP 
      t_NumberOfActiveSteps : Int;
   END_VAR


BEGIN
	  
	  #t_NumberOfActiveSteps := #InOutG7Arrays[#InOutRTData.OFFSETS.SAX_OFFSET] - 1;
	  
	  
END_FUNCTION_BLOCK
